TYPE T_Ctrl_SIf_ICL_Par:
STRUCT
	Module: T_Ctrl_SIf_MOD_Par;
END_STRUCT
END_TYPE

(* stored: Version 1.1.0.1, ProductVersion 3.1.0.19
   DUT T_Ctrl_SIf_ICL_Par: Id {f4d3cf1c-1d6c-40ce-b959-82e6fd131622} *)
